(*
Worker wrapper that runs job until completition.
*)
FUNCTION_BLOCK BlockingWorker
VAR
	_scheduler: Worker;
END_VAR

(*
Returns internal Worker.
*)
PROPERTY Base : I_Worker
GET
Base := _scheduler;
END_GET
END_PROPERTY

METHOD Run
VAR_INPUT
END_VAR
IF _scheduler.First = 0 THEN
	RETURN;
END_IF

CASE _scheduler.First.State OF
	JobState.Completed, JobState.Aborted:
		_scheduler.Dequeue(_scheduler.First);
END_CASE

CASE _scheduler.Run(_scheduler.First) OF
	Ok:
		// Do Nothing
	Err.Itf0:
		RETURN;
	ELSE
		DebugMsg(_scheduler, 'Scheduler: Incorrect task state!');
		DebugMsg(_scheduler.First, 'Task: Incorrect task state!');
		RETURN;	
END_CASE
END_METHOD

END_FUNCTION_BLOCK

(* stored: Version 1.1.0.1
   POU BlockingWorker: Id {4df31f95-b8c5-4f13-a754-0d5e2a3c4dcf}, SpecialFunc None
   Property Base: Id {428f8038-c731-4fcf-8d16-6aea864f3d2f}
   Get Get: Id {d8fdf29e-8280-45d4-aace-254a56c73568}
   Method Run: Id {b01bdd15-c311-4810-9031-f686d33604bb} *)
